(*******************************************************************************
 * Interface: I_Syntax_ExhaustiveComments
 * Description: Interface with doc comments and parameter comments.
 *******************************************************************************)
INTERFACE I_Syntax_ExhaustiveComments EXTENDS __SYSTEM.IQueryInterface

/// <summary>Executes a device command.</summary>
METHOD ExecuteCommand : BOOL
VAR_INPUT
    nCmdId : DINT; (* Command identifier *)
    fParam : LREAL; // Command parameter value
END_VAR
VAR_OUTPUT
    nStatus : UDINT; (* Result status code *)
END_VAR
END_METHOD

/// <summary>True when device is ready.</summary>
PROPERTY P_Operational : BOOL
GET
END_GET
END_PROPERTY

END_INTERFACE

(* stored: Version 1.1.0.1, ProductVersion 3.1.4024.16
   Itf I_Syntax_ExhaustiveComments: Id {04b92435-2295-4863-8358-e8cfc52a4b25}
   Method ExecuteCommand: Id {e2a49e42-99b4-48c9-a149-042046df65ef}
   Property P_Operational: Id {94fb8abc-6a0f-428b-b1d4-841267d6148b}
   Get Get: Id {11809c1f-fb9e-4194-886d-5f89d4e34ddc} *)
